TYPE ST_MotionParameters :
STRUCT
END_STRUCT
END_TYPE

(* stored: Version 1.1.0.1, ProductVersion 3.1.4024.12
   DUT ST_MotionParameters: Id {4cdb79a0-4b29-4b4c-91d1-feba1705b6b2} *)
